FUNCTION_BLOCK FB_PNEUMATIC_AXIS
VAR_INPUT
    stPneumaticAxisInputs: ST_PneumaticAxisInputs;
    stPneumaticAxisControl: ST_PneumaticAxisControl;
 END_VAR

VAR_OUTPUT
    stPneumaticAxisStatus: ST_PneumaticAxisStatus;
END_VAR

VAR
    ePneumaticAxisState: E_PneumaticMode;
    fbTimerExtend: TON; //Timing the extraction of the cylinder
    fbTimerRetract: TON; //Timing the retraction of the cylinder
    fbTimerExtendManual: TON; //Timing the extraction of the cylinder
    fbTimerRetractManual: TON; //Timing the retraction of the cylinder
    bStateChange: BOOL := FALSE; //State of the cylinder changed from extend to retract and vice versa

END_VAR

//Single solenoid valve control
//Starting the extraction movement and extraction timing
//LimitBwd is activated and cylinder is not extracted

CASE ePneumaticAxisState OF
    E_PneumaticMode.SINGLE_SOLENOID_PLC:
        IF (stPneumaticAxisControl.bStartExtend AND stPneumaticAxisInputs.bPermit) AND NOT stPneumaticAxisInputs.bLimitFwd THEN
        stPneumaticAxisStatus.bExtendMoving := TRUE;
        stPneumaticAxisStatus.bMoving := TRUE;
        fbTimerExtend (IN := stPneumaticAxisStatus.bExtendMoving, PT := T#20S);
        IF fbTimerExtend.Q THEN
            ePneumaticAxisState := E_PneumaticMode.ERROR;
        END_IF
    END_IF

// Extraction of the cylinder finished, reset timer
        IF stPneumaticAxisInputs.bLimitFwd AND NOT stPneumaticAxisInputs.bLimitBwd THEN
        stPneumaticAxisStatus.sStatus := 'EXTRACTED';
        stPneumaticAxisStatus.bExtracted := TRUE;
        bStateChange := TRUE;
        stPneumaticAxisStatus.bExtendMoving := FALSE;
        stPneumaticAxisStatus.bMoving := FALSE;
        fbTimerExtend (IN := stPneumaticAxisStatus.bExtendMoving, PT := T#20S);
    END_IF

//Starting the retraction movement and retraction timing
        IF NOT stPneumaticAxisControl.bStartExtend AND NOT stPneumaticAxisInputs.bLimitBwd AND bStateChange THEN
        stPneumaticAxisStatus.bRetractMoving := TRUE;
        stPneumaticAxisStatus.bMoving := TRUE;
        stPneumaticAxisStatus.bExtracted := FALSE;
        fbTimerRetract (IN := stPneumaticAxisStatus.bRetractMoving, PT := T#20S);
        IF fbTimerRetract.Q THEN
            ePneumaticAxisState := E_PneumaticMode.ERROR;
        END_IF
    END_IF

// Retraction of the cylinder finished, reset timer
        IF NOT stPneumaticAxisControl.bStartExtend AND stPneumaticAxisInputs.bLimitBwd THEN
        stPneumaticAxisStatus.sStatus := 'RETRACTED';
        stPneumaticAxisStatus.bRetracted := TRUE;
        bStateChange := FALSE;
        stPneumaticAxisStatus.bRetractMoving := FALSE;
        stPneumaticAxisStatus.bMoving := FALSE;
        fbTimerRetract (IN := stPneumaticAxisStatus.bRetractMoving, PT := T#20S);
     END_IF


        E_PneumaticMode.SINGLE_SOLENOID_MANUAL:
//Manual control of single solenoid pneumatic actuator
//Extend cylinder
        IF stPneumaticAxisInputs.bExtendCylinderManual AND NOT stPneumaticAxisInputs.bLimitFwd THEN
        stPneumaticAxisStatus.bExtendMoving := TRUE;
        fbTimerExtendManual (IN := stPneumaticAxisStatus.bExtendMoving, PT := T#20S);
        IF fbTimerExtendManual.Q THEN
            ePneumaticAxisState := E_PneumaticMode.ERROR;
        END_IF
    END_IF

//Extraction of the cylinder finished, reset timer
        IF stPneumaticAxisInputs.bLimitFwd THEN
        stPneumaticAxisStatus.sStatus := 'EXTRACTED';
        bStateChange := TRUE;
        stPneumaticAxisStatus.bExtendMoving := FALSE;
        fbTimerExtendManual (IN := stPneumaticAxisStatus.bExtendMoving, PT := T#20S);
    END_IF

//Starting the retraction movement and extraction timing
        IF stPneumaticAxisInputs.bRetractCylinderManual AND NOT stPneumaticAxisInputs.bLimitBwd AND bStateChange THEN
        stPneumaticAxisInputs.bExtendCylinderManual := FALSE;
        stPneumaticAxisStatus.bRetractMoving := TRUE;
        fbTimerRetractManual (IN := stPneumaticAxisStatus.bRetractMoving, PT := T#20S);
        IF fbTimerRetractManual.Q THEN
            ePneumaticAxisState := E_PneumaticMode.ERROR;
        END_IF
    END_IF

//Retraction of the cylinder finished, reset timer
        IF stPneumaticAxisInputs.bLimitBwd THEN
        stPneumaticAxisStatus.sStatus := 'RETRACTED';
        bStateChange := FALSE;
        stPneumaticAxisStatus.bRetractMoving := FALSE;
        fbTimerRetractManual (IN := stPneumaticAxisStatus.bRetractMoving, PT := T#20S);
        stPneumaticAxisInputs.bRetractCylinderManual := FALSE;
    END_IF

    E_PneumaticMode.ERROR:
    stPneumaticAxisStatus.sStatus := 'ERROR: COMMAND TIMED OUT';

    E_PneumaticMode.RESET:
    stPneumaticAxisControl.bStartExtend := FALSE;
    stPneumaticAxisInputs.bExtendCylinderManual := FALSE;
    fbTimerExtend.IN := FALSE;
    fbTimerRetract.IN := FALSE;
    fbTimerExtendManual.IN := FALSE;
    fbTimerRetractManual.IN := FALSE;
END_CASE

ACTION Single_Solenoid:

END_ACTION

END_FUNCTION_BLOCK

(* stored: Version 1.1.0.1, ProductVersion 3.1.4024.5
   POU FB_PNEUMATIC_AXIS: Id {74b90e1e-7e39-4d6d-a9f3-f7a29858f68b}, SpecialFunc None
   Action Single_Solenoid: Id {a75a03ea-ec30-403c-91eb-96684f17a503} *)
